{region '#Template'}
	{attribute 'Version' := '5.0.0.0'}
	{attribute 'Tags' := '"LCID": "1031", "Text": "AC, Allgemein, AHU, Sequenz, Sequenzverbindung, Temperatur"'}
	{attribute 'Tags' := '"LCID": "1033", "Text": "AC, General, AHU, Sequence, Sequence link, Temperature"'}
	{attribute 'Using' := '"Type": "Template", "URI": "E_BA_AC_OpMod01"'}
	{attribute 'Using' := '"Type": "Template", "URI": "E_AC_SeqNumber_T"'}
	{attribute 'Description' := '"LCID": "1031", "Text": "Sequenzverbindung"'}
	{attribute 'Description' := '"LCID": "1033", "Text": "Sequence link"'}
{endregion}

FUNCTION_BLOCK FB_BA_AC_SeqT EXTENDS FB_BA_View
VAR_INPUT
	bEn					: BOOL;
	eOpMode				: E_BA_AC_OpMod01;		
	fTWth				: REAL;
END_VAR
VAR_OUTPUT
	bSumLmt				: BOOL;		//Sommer Grenzwert ist aktiv	//	Summer limit is active
	bWinLmt				: BOOL;		//Winter Grenzwert ist aktiv	//	Winter limit is active
	nActvSeqCtrl		: UDINT;	// Nummer des aktiven Sequenzcontrollers // number of the active sequenz controller
END_VAR
VAR_IN_OUT
	stTSeqLink			: ST_BA_SeqLink;	//	Sequenz Link Struktur	//	Sequence link structure	
END_VAR
VAR_INPUT CONSTANT
	WthTLmtSum			: FB_BA_AV_Op;
	WthTLmtWin			: FB_BA_AV_Op;
	SeqLink				: FB_BA_SequenceLinkBase;		//	Hauptprogramm zur Steuerung der Sequenzregler einer Anlage	//	Main program to control the sequence controller of a plant
	ActvSeqCtrl			: FB_BA_MV_Op;	
END_VAR
VAR
	WthTLmtWinHys		: FB_BA_Swi2P;			//	Hysterese Grenzwert Winter									//	Hysteresis limit winter
	WthTLmtSumHys		: FB_BA_Swi2P;			//	Hysterese Grenzwert Sommer									//	Hysteresis limit summer
	StartSeq			: FB_BA_PrioSwi_UDI08;	//	Festlegung Start Sequenz									//	Fixing start-up sequence
END_VAR

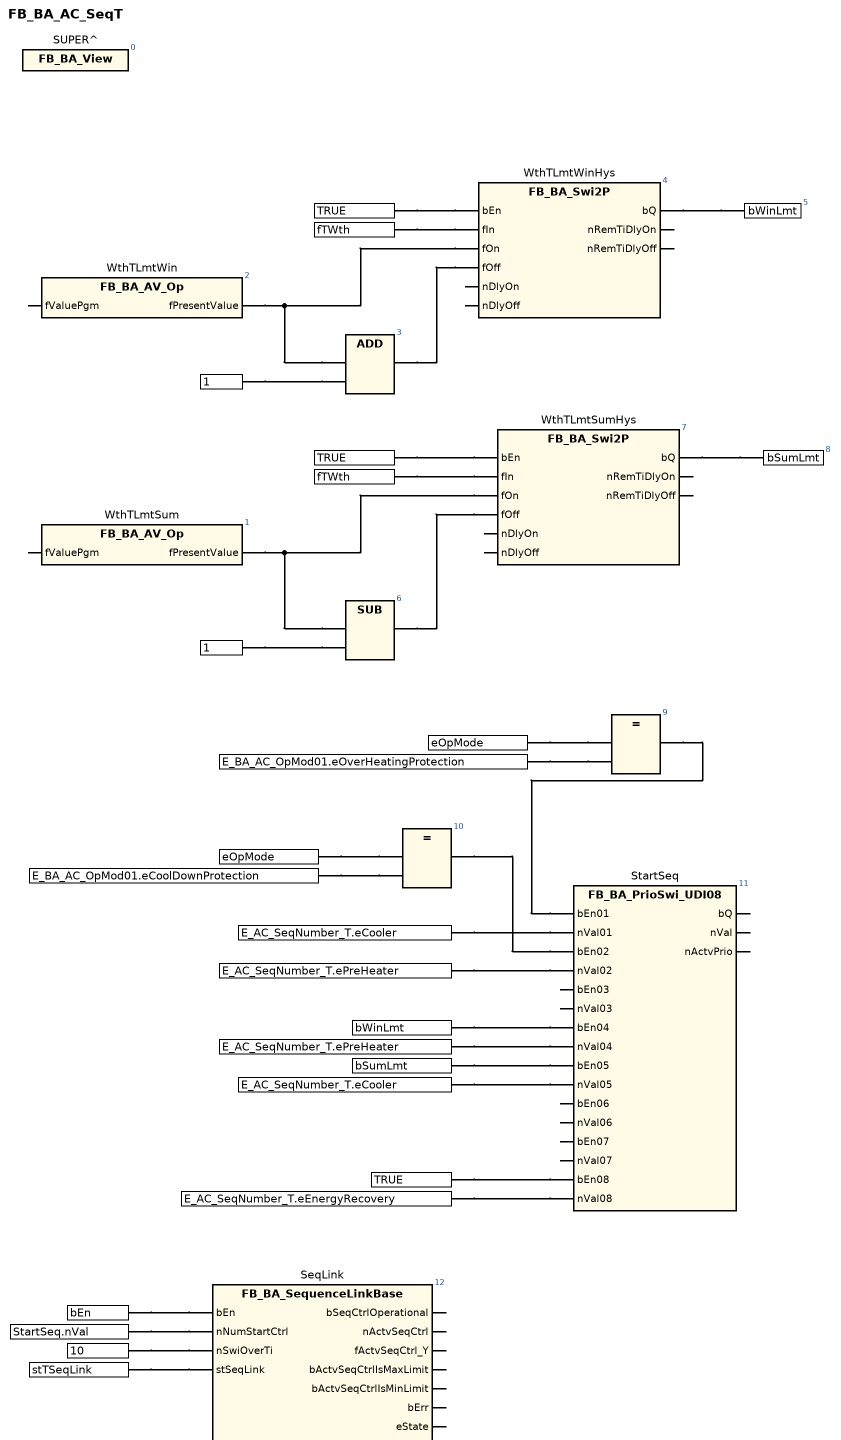
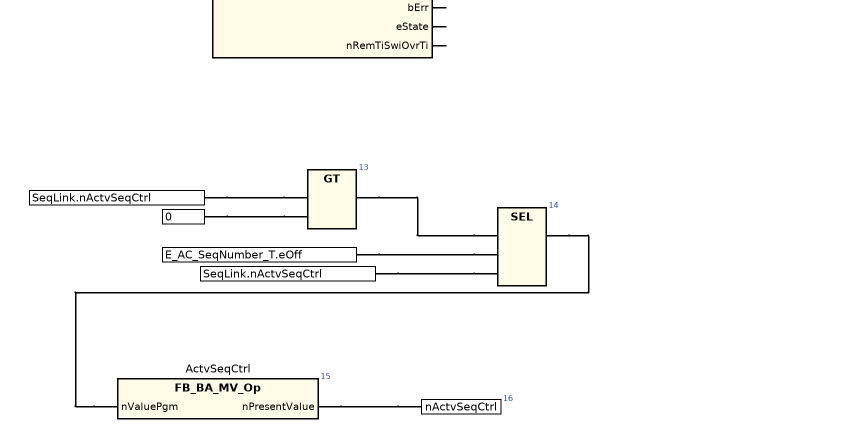
SUPER^(); // FB_BA_View
WthTLmtSum(); // FB_BA_AV_Op
WthTLmtWin(); // FB_BA_AV_Op
WthTLmtWinHys(
    bEn := TRUE,
    fIn := fTWth,
    fOn := WthTLmtWin.fPresentValue,
    fOff := WthTLmtWin.fPresentValue + 1); // FB_BA_Swi2P
bWinLmt := WthTLmtWinHys.bQ;
WthTLmtSumHys(
    bEn := TRUE,
    fIn := fTWth,
    fOn := WthTLmtSum.fPresentValue,
    fOff := WthTLmtSum.fPresentValue - 1); // FB_BA_Swi2P
bSumLmt := WthTLmtSumHys.bQ;
StartSeq(
    bEn01 := eOpMode = E_BA_AC_OpMod01.eOverHeatingProtection,
    nVal01 := E_AC_SeqNumber_T.eCooler,
    bEn02 := eOpMode = E_BA_AC_OpMod01.eCoolDownProtection,
    nVal02 := E_AC_SeqNumber_T.ePreHeater,
    bEn04 := bWinLmt,
    nVal04 := E_AC_SeqNumber_T.ePreHeater,
    bEn05 := bSumLmt,
    nVal05 := E_AC_SeqNumber_T.eCooler,
    bEn08 := TRUE,
    nVal08 := E_AC_SeqNumber_T.eEnergyRecovery); // FB_BA_PrioSwi_UDI08
SeqLink(bEn := bEn, nNumStartCtrl := StartSeq.nVal, nSwiOverTi := 10, stSeqLink := stTSeqLink); // FB_BA_SequenceLinkBase
ActvSeqCtrl(nValuePgm := SEL(SeqLink.nActvSeqCtrl > 0, E_AC_SeqNumber_T.eOff, SeqLink.nActvSeqCtrl)); // FB_BA_MV_Op
nActvSeqCtrl := ActvSeqCtrl.nPresentValue;

METHOD FB_init : BOOL
VAR_INPUT
	bInitRetains : BOOL; // if TRUE, the retain variables are initialized (warm start / cold start)
	bInCopyCode : BOOL;  // if TRUE, the instance afterwards gets moved into the copy code (online change)
END_VAR
WthTLmtSum.iParent							:= THIS^;
WthTLmtSum.iLabel							:= LblCtl_LimitValueWeatherTemperatureSummer;
WthTLmtSum.eUnit 							:= E_BA_Unit.eTemperature_DegreesCelsius;								 
WthTLmtSum.fValueRm							:= 10;	
WthTLmtSum.fCOVIncrement					:= BA2_Param.fDefCOVIncrement;		

WthTLmtWin.iParent							:= THIS^;
WthTLmtWin.iLabel							:= LblCtl_LimitValueWeatherTemperatureWinter;
WthTLmtWin.eUnit 							:= E_BA_Unit.eTemperature_DegreesCelsius;								 
WthTLmtWin.fValueRm							:= 20;	
WthTLmtWin.fCOVIncrement					:= BA2_Param.fDefCOVIncrement;		

SeqLink.fHys								:= 2;
SeqLink.eNoStartCtrlFound					:= E_BA_NoStartCtrlFound.eLastActionReverse;	
SeqLink.eNoEnableSeqCtrl					:= E_BA_NoEnableSeqCtrl.eNextAction;	

ActvSeqCtrl.iParent							:= THIS^;
ActvSeqCtrl.iLabel							:= LblCtl_CurrentSequenceTemperature;
ActvSeqCtrl.aStateText[1]					:= txtEvent_Reheater;
ActvSeqCtrl.aStateText[2]					:= txtEvent_Preheater;
ActvSeqCtrl.aStateText[3]					:= txtEvent_MixedAir;
ActvSeqCtrl.aStateText[4]					:= txtEvent_EnergyRecovery;
ActvSeqCtrl.aStateText[5]					:= txtEvent_Cooler;
ActvSeqCtrl.aStateText[6]					:= txtEvent_Off;
END_METHOD

END_FUNCTION_BLOCK

(* stored: Version 1.1.0.1, ProductVersion 3.1.4024.12
   POU FB_BA_AC_SeqT: Id {72ec69c7-e923-4067-be79-442f9f8d48cd}, SpecialFunc None
   Method FB_init: Id {ac33d490-b453-4d93-ba53-84a70954abfd} *)
